Universal Robots PolyScope program: Wheel.urp

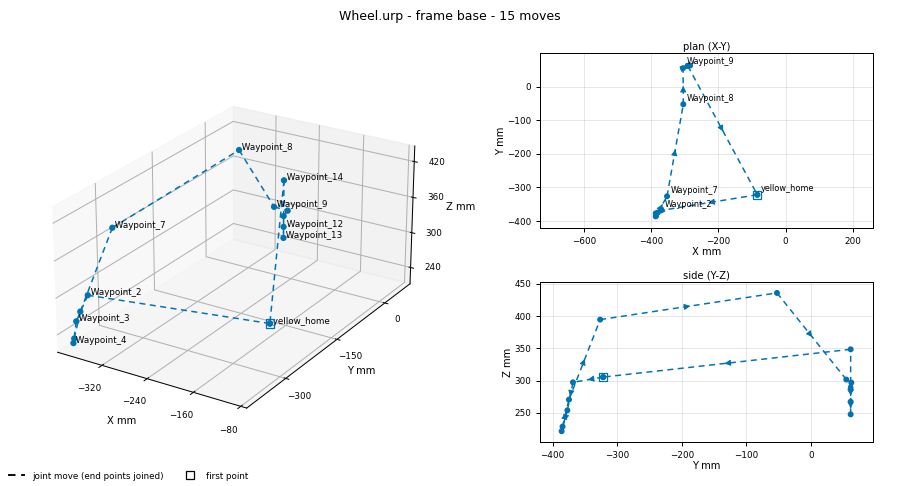
[picture p0: tool path of Wheel.urp in frame base, 15 of 15 moves have a stored position in this frame; points joined in program order, loops and branches not executed]
Program Wheel (installation=default directory=/programs/usbdisk/Zahra1 createdIn=5.11.11.1010533 lastSavedIn=5.11.11.1010533 robotSerialNumber=20205300864)
Calibrated DH parameters: a=[-0.000166, -0.243494, -0.153108, 0.000057, -0.000123, 0]; d=[0.151897, -1.34267, 53.988124, -52.514559, 0.085283, 0.092193]; alpha=[1.572472, -0.003756, 0.002824, 1.570807, -1.572621, 0]; deltaTheta=[0, 0.020704, 7.033215, -0.770746, 0.000004, 0]
Robot Program (runOnlyOnce=true)
  MoveJ speed 60 deg/s, acceleration 80 deg/s^2 (useActiveTCP=true) feature=Base
    Waypoint yellow_home: TCP in base x=-84.299 y=-321.875 z=305.481 mm, rx=-2.0809 ry=-2.2572 rz=0.0984 rad; joints [-79.978, -91.201, -87.971, -91.7, 84.671, 815.506] deg
    URCap Gripper (Robotiq_Grippers, Robotiq Inc.) dataModel(position=25.098039215686274, force=94.0, speed=40.0, positionInDouble=25.098039215686274, forceInDouble=94.0, speedInDouble=40.0, slaveIds=[9], blocking=true, robotCompliant=false)
    Waypoint Waypoint_2: TCP in base x=-370.284 y=-368.602 z=297.382 mm, rx=-2.0396 ry=-2.1945 rz=0.3804 rad; joints [-118.722, -144.818, -14.422, -98.204, 79.573, 775.887] deg
    Waypoint Waypoint_3: TCP in base x=-386.489 y=-377.29 z=253.992 mm, rx=-2.2315 ry=-2.101 rz=0.3689 rad; joints [-120.441, -150.431, -15.095, -92.007, 83.012, 782.191] deg
    Waypoint Waypoint_4: TCP in base x=-386.472 y=-386.16 z=221.689 mm, rx=-2.1674 ry=-2.1413 rz=0.2909 rad; joints [-119.861, -154.029, -15.223, -91.317, 82.455, 780.154] deg
    URCap Gripper (Robotiq_Grippers, Robotiq Inc.) dataModel(position=94.41176470588235, force=94.0, speed=40.0, positionInDouble=94.41176470588235, forceInDouble=94.0, speedInDouble=40.0, slaveIds=[9], blocking=true, robotCompliant=false)
    Waypoint Waypoint_5: TCP in base x=-385.798 y=-384.764 z=228.778 mm, rx=-2.1687 ry=-2.1411 rz=0.3034 rad; joints [-119.87, -153.218, -15.166, -91.706, 82.446, 780.15] deg
    Waypoint Waypoint_6: TCP in base x=-380.3 y=-374.811 z=270.634 mm, rx=-2.1458 ry=-2.1723 rz=0.3765 rad; joints [-119.927, -148.234, -15.089, -93.853, 82.686, 778.493] deg
    Waypoint Waypoint_7: TCP in base x=-352.792 y=-326.487 z=394.487 mm, rx=-2.1584 ry=-2.1624 rz=0.6193 rad; joints [-119.929, -134.878, -9.798, -103.32, 82.69, 778.493] deg
    Waypoint Waypoint_8: TCP in base x=-304.391 y=-52.738 z=435.766 mm, rx=3.1003 ry=0.0056 rz=-0.1159 rad; joints [-144.9, -93.309, -50.695, -121.099, 89.301, 844.916] deg
    Waypoint Waypoint_9: TCP in base x=-305.124 y=54.628 z=301.671 mm, rx=-3.1176 ry=0.0327 rz=-0.0279 rad; joints [-164.928, -86.198, -93.63, -91.424, 89.01, 826.384] deg
    Waypoint Waypoint_10: TCP in base x=-284.251 y=62.458 z=296.857 mm, rx=-3.1128 ry=0.083 rz=0.087 rad; joints [-164.925, -79.454, -102.353, -85.458, 87.694, 828.175] deg
    Waypoint Waypoint_11: TCP in base x=-291.02 y=61.356 z=286.286 mm, rx=-3.0968 ry=0.0814 rz=0.0417 rad; joints [-164.921, -81.889, -102.446, -84.798, 87.236, 828.177] deg
    Waypoint Waypoint_12: TCP in base x=-291.012 y=61.362 z=267.326 mm, rx=-3.0969 ry=0.0815 rz=0.0415 rad; joints [-164.931, -82.445, -107.109, -79.583, 87.249, 828.183] deg
    Waypoint Waypoint_13: TCP in base x=-291.011 y=61.359 z=247.779 mm, rx=-3.0969 ry=0.0815 rz=0.0415 rad; joints [-164.939, -83.482, -111.596, -74.059, 87.256, 828.189] deg
    URCap Gripper (Robotiq_Grippers, Robotiq Inc.) dataModel(position=21.176470588235293, force=70.0, speed=67.0, positionInDouble=21.176470588235293, forceInDouble=70.0, speedInDouble=67.0, slaveIds=[9], blocking=true, robotCompliant=false)
    Waypoint Waypoint_14: TCP in base x=-291.009 y=61.367 z=348.473 mm, rx=-3.0969 ry=0.0815 rz=0.0415 rad; joints [-164.898, -82.914, -84.757, -101.465, 87.206, 828.173] deg
    Waypoint yellow_home: TCP in base x=-84.299 y=-321.875 z=305.481 mm, rx=-2.0809 ry=-2.2572 rz=0.0984 rad; joints [-79.978, -91.201, -87.971, -91.7, 84.671, 815.506] deg
